(* IEC 61131-3 sources: hello-ax-world/src, 3 files *)

(* ---- HelloWorldFunction.st ---- *)
NAMESPACE Siemens.Ax
    FUNCTION HelloWorldFunction : STRING
        HelloWorldFunction := 'Hello AX World';
    END_FUNCTION
END_NAMESPACE

(* ---- configuration.st ---- *)
CONFIGURATION MyConfiguration
    // Create main task
    TASK Main(Priority := 1);

    // Assign MyProgram to main (cyclic) task
    PROGRAM P1 WITH Main: MyProgram;

    VAR_GLOBAL
        myString : String := 'Hello World';
    END_VAR

END_CONFIGURATION

(* ---- program.st ---- *)
PROGRAM MyProgram
    VAR_EXTERNAL
        myString : String;
    END_VAR

    VAR

    END_VAR

    VAR_TEMP

    END_VAR

    myString := Siemens.Ax.HelloWorldFunction();

END_PROGRAM
